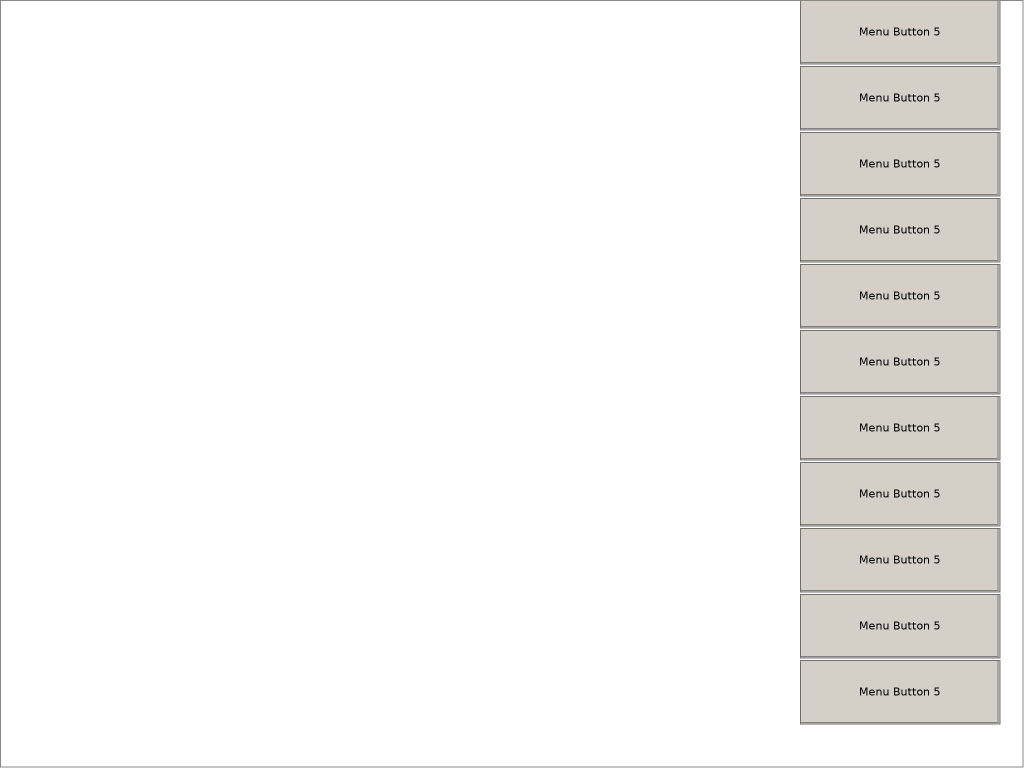
VISUALIZATION PopupMenu5  // 1024x768
    Button (800,0 200x64), "Menu Button 5"
        OnMouseClick: CloseDialog Dialog=PopupMenu5, Result=None, NumpadKeypadSet=True
    Button (800,66 200x64), "Menu Button 5"
        OnMouseClick: CloseDialog Dialog=PopupMenu5, Result=None, NumpadKeypadSet=True
    Button (800,132 200x64), "Menu Button 5"
        OnMouseClick: CloseDialog Dialog=PopupMenu5, Result=None, NumpadKeypadSet=True
    Button (800,198 200x64), "Menu Button 5"
        OnMouseClick: CloseDialog Dialog=PopupMenu5, Result=None, NumpadKeypadSet=True
    Button (800,264 200x64), "Menu Button 5"
        OnMouseClick: CloseDialog Dialog=PopupMenu5, Result=None, NumpadKeypadSet=True
    Button (800,330 200x64), "Menu Button 5"
        OnMouseClick: CloseDialog Dialog=PopupMenu5, Result=None, NumpadKeypadSet=True
    Button (800,396 200x64), "Menu Button 5"
        OnMouseClick: CloseDialog Dialog=PopupMenu5, Result=None, NumpadKeypadSet=True
    Button (800,462 200x64), "Menu Button 5"
        OnMouseClick: CloseDialog Dialog=PopupMenu5, Result=None, NumpadKeypadSet=True
    Button (800,528 200x64), "Menu Button 5"
        OnMouseClick: CloseDialog Dialog=PopupMenu5, Result=None, NumpadKeypadSet=True
    Button (800,594 200x64), "Menu Button 5"
        OnMouseClick: CloseDialog Dialog=PopupMenu5, Result=None, NumpadKeypadSet=True
    Button (800,660 200x64), "Menu Button 5"
        OnMouseClick: CloseDialog Dialog=PopupMenu5, Result=None, NumpadKeypadSet=True
    InvisibleInput (1000,0 25x768)
        OnMouseClick: CloseDialog Dialog=PopupMenu5, Result=Cancel, NumpadKeypadSet=True
    InvisibleInput (0,0 800x768)
        OnMouseClick: CloseDialog Dialog=PopupMenu5, Result=OK, NumpadKeypadSet=True
    InvisibleInput (800,726 203x44)
        OnMouseClick: CloseDialog Dialog=PopupMenu5, Result=Cancel, NumpadKeypadSet=True
END_VISUALIZATION

(* stored: Version 1.1.0.1, ProductVersion 3.1.4024.11
   Visu PopupMenu5: Id {95648dc3-dcd5-0a86-03ea-0ef75f84d4f8} *)
